FUNCTION_BLOCK PUBLIC FB_MusicStopCommand IMPLEMENTS I_Command
VAR
	refCDPlayer : REFERENCE TO FB_CDPlayer;
END_VAR

METHOD Execute
IF (__ISVALIDREF(THIS^.refCDPlayer)) THEN
	THIS^.refCDPlayer.Stop();
END_IF
END_METHOD

METHOD FB_init : BOOL
VAR_INPUT
	bInitRetains : BOOL; // if TRUE, the retain variables are initialized (warm start / cold start)
	bInCopyCode : BOOL;  // if TRUE, the instance afterwards gets moved into the copy code (online change)
	refCDPlayer : REFERENCE TO FB_CDPlayer;
END_VAR
IF (__ISVALIDREF(refCDPlayer)) THEN
	THIS^.refCDPlayer REF= refCDPlayer;
ELSE
	THIS^.refCDPlayer REF= 0;
END_IF
END_METHOD

METHOD Undo
IF (__ISVALIDREF(THIS^.refCDPlayer)) THEN
	THIS^.refCDPlayer.SetVolume(40);
	THIS^.refCDPlayer.SetTrack(1);
	THIS^.refCDPlayer.Start();
END_IF
END_METHOD

END_FUNCTION_BLOCK

(* stored: Version 1.1.0.1, ProductVersion 3.1.4020.3
   POU FB_MusicStopCommand: Id {8cf03a18-b11f-47a4-bd12-bfcb0a33580c}, SpecialFunc None
   Method Execute: Id {86d54cc1-f415-4974-832c-25dca3ebebfb}
   Method FB_init: Id {15f8b24f-95fe-4769-b3bd-5a189cb73ec8}
   Method Undo: Id {bdee52f1-1b95-4630-81e4-a5e10d4b74cb} *)
